{attribute 'GeneratedUsingTerminal: CU1123-0000-0016'}
{attribute addProperty BoxType "CU1123-0000-0016"}
{attribute addProperty Id "A_0002_CU1123_0010_0016A_0002_CU1123_0010_0016_E2D71E5192"}
{attribute addProperty CRC "126784336"}
{attribute addProperty Size "92"}
TYPE A_0001_CU1123_0000_0016_078E9350 EXTENDS CU1123_1FC0878B :
STRUCT
	{attribute addProperty Name "A_0002_CU1123_0010_0016"}
	{attribute addProperty PreviousPort "A_0001(CU1123-0000-0016) : D"}
	A_0002_CU1123_0010_0016 : A_0002_CU1123_0010_0016_E2D71E51;
END_STRUCT
END_TYPE

(* stored: Version 1.2.0.0, ProductVersion 3.1.4024.9
   DUT A_0001_CU1123_0000_0016_078E9350: Id {505bfa66-5337-4f39-b978-bd82f0b67a05} *)
